// TIA Portal V17 export
// export: Created 2021-12-03T08:12:59.6189284Z, ExportSetting WithDefaults, DisplayName Totally Integrated Automation Portal, DisplayVersion V17, DisplayName TIA Portal Openness, DisplayVersion V17, DisplayName TIA Portal Version Control Interface, DisplayVersion V17, DisplayName STEP 7 Professional, DisplayVersion V17, DisplayName STEP 7 Safety, DisplayVersion V17, DisplayName WinCC Advanced, DisplayVersion V17
FUNCTION_BLOCK "FB_ScanSequence"   // FB70, GRAPH
VERSION : 0.1
// stored: AcknowledgeErrorsRequired true, AutoNumber false, CreateMinimizedDB false, IsIECCheckEnabled false, LanguageInNetworks LAD, LockOperatingMode false, PermanentILProcessingInMANMode false, SkipSteps false, UDAEnableTagReadback false, WithAlarmHandling true
   VAR_INPUT
      OFF_SQ { ExternalAccessible := 'False'; ExternalVisible := 'False'; ExternalWritable := 'False'} : Bool := false;   // Turn sequence off
      INIT_SQ { ExternalAccessible := 'False'; ExternalVisible := 'False'; ExternalWritable := 'False'} : Bool := false;   // Set sequence to initial state
      ACK_EF { ExternalAccessible := 'False'; ExternalVisible := 'False'; ExternalWritable := 'False'} : Bool := false;   // Acknowledge all errors and faults
      S_PREV { ExternalAccessible := 'False'; ExternalVisible := 'False'; ExternalWritable := 'False'} : Bool := false;   // Output previous step in parameter S_NO
      S_NEXT { ExternalAccessible := 'False'; ExternalVisible := 'False'; ExternalWritable := 'False'} : Bool := false;   // Indicate next step in parameter S_NO
      SW_AUTO { ExternalAccessible := 'False'; ExternalVisible := 'False'; ExternalWritable := 'False'} : Bool := false;   // Automatic mode
      SW_TAP { ExternalAccessible := 'False'; ExternalVisible := 'False'; ExternalWritable := 'False'} : Bool := false;   // Semiautomatic/switch with transition
      SW_TOP { ExternalAccessible := 'False'; ExternalVisible := 'False'; ExternalWritable := 'False'} : Bool := false;   // Semiautomatic/ignore transition
      SW_MAN { ExternalAccessible := 'False'; ExternalVisible := 'False'; ExternalWritable := 'False'} : Bool := false;   // Manual mode
      S_SEL { ExternalAccessible := 'False'; ExternalVisible := 'False'; ExternalWritable := 'False'} : Int := 0;   // Select step to be output to S_NO
      S_ON { ExternalAccessible := 'False'; ExternalVisible := 'False'; ExternalWritable := 'False'} : Bool := false;   // Activate step indicated in S_NO
      S_OFF { ExternalAccessible := 'False'; ExternalVisible := 'False'; ExternalWritable := 'False'} : Bool := false;   // Deactivate step indicated S_NO
      T_PUSH { ExternalAccessible := 'False'; ExternalVisible := 'False'; ExternalWritable := 'False'} : Bool := false;   // Enable transition to switch in semi automatic mode
   END_VAR
   VAR_OUTPUT
      S_NO { ExternalAccessible := 'False'; ExternalVisible := 'False'; ExternalWritable := 'False'} : Int := 0;   // Step number
      S_MORE { ExternalAccessible := 'False'; ExternalVisible := 'False'; ExternalWritable := 'False'} : Bool := false;   // More steps are available and can be shown in S_NO
      S_ACTIVE { ExternalAccessible := 'False'; ExternalVisible := 'False'; ExternalWritable := 'False'} : Bool := false;   // Step indicated in S_NO is active
      ERR_FLT { ExternalAccessible := 'False'; ExternalVisible := 'False'; ExternalWritable := 'False'} : Bool := false;   // Interlock or supervision group error
      AUTO_ON { ExternalAccessible := 'False'; ExternalVisible := 'False'; ExternalWritable := 'False'} : Bool := false;   // Automatic mode is active
      TAP_ON { ExternalAccessible := 'False'; ExternalVisible := 'False'; ExternalWritable := 'False'} : Bool := false;   // Semiautomatic mode/step with transition enabled
      TOP_ON { ExternalAccessible := 'False'; ExternalVisible := 'False'; ExternalWritable := 'False'} : Bool := false;   // Semiautomatic mode/ignore transition enabled
      MAN_ON { ExternalAccessible := 'False'; ExternalVisible := 'False'; ExternalWritable := 'False'} : Bool := false;   // Manual mode is active
   END_VAR
   VAR DB_SPECIFIC
      S_DISPLAY { ExternalAccessible := 'False'; ExternalVisible := 'False'; ExternalWritable := 'False'} : Int;   // Internal display of output parameter S_NO
      S_SEL_OLD { ExternalAccessible := 'False'; ExternalVisible := 'False'; ExternalWritable := 'False'} : Int;   // Previous value in S_SEL
      S_DISPIDX { ExternalAccessible := 'False'; ExternalVisible := 'False'; ExternalWritable := 'False'} : Byte;   // Index of the step in S_NO
      T_DISPIDX { ExternalAccessible := 'False'; ExternalVisible := 'False'; ExternalWritable := 'False'} : Byte;   // Index of the transition displayed in T_NO
      MOP { ExternalAccessible := 'False'; ExternalVisible := 'False'; ExternalWritable := 'False'} : Struct   // Mode
         AUTO { ExternalAccessible := 'False'; ExternalVisible := 'False'; ExternalWritable := 'False'} : Bool := true;   // Status: automatic mode
         MAN { ExternalAccessible := 'False'; ExternalVisible := 'False'; ExternalWritable := 'False'} : Bool := false;   // Status: manual mode
         TAP { ExternalAccessible := 'False'; ExternalVisible := 'False'; ExternalWritable := 'False'} : Bool := false;   // Status: semi automatic/switch with transition
         TOP { ExternalAccessible := 'False'; ExternalVisible := 'False'; ExternalWritable := 'False'} : Bool := false;   // Status: semi automatic/ignore transition
         ACK_S { ExternalAccessible := 'False'; ExternalVisible := 'False'; ExternalWritable := 'False'} : Bool := false;   // Request: acknowledge step at parameter S_NO
         REG_S { ExternalAccessible := 'False'; ExternalVisible := 'False'; ExternalWritable := 'False'} : Bool := false;   // Request: register step indicated in S_NO
         T_PREV { ExternalAccessible := 'False'; ExternalVisible := 'False'; ExternalWritable := 'False'} : Bool := false;   // Request: output previous valid transition in T_NO
         T_NEXT { ExternalAccessible := 'False'; ExternalVisible := 'False'; ExternalWritable := 'False'} : Bool := false;   // Request: output next valid transition in T_NO
         LOCK { ExternalAccessible := 'False'; ExternalVisible := 'False'; ExternalWritable := 'False'} : Bool := true;   // Status: interlocks activated
         SUP { ExternalAccessible := 'False'; ExternalVisible := 'False'; ExternalWritable := 'False'} : Bool := true;   // Status: supervisions activated
         ACKREQ { ExternalAccessible := 'False'; ExternalVisible := 'False'; ExternalWritable := 'False'} : Bool := true;   // Status: acknowledgment required
         SSKIP { ExternalAccessible := 'False'; ExternalVisible := 'False'; ExternalWritable := 'False'} : Bool := false;   // Status: "Skip steps" enabled
         OFF { ExternalAccessible := 'False'; ExternalVisible := 'False'; ExternalWritable := 'False'} : Bool := false;   // Request: deactivate all steps
         INIT { ExternalAccessible := 'False'; ExternalVisible := 'False'; ExternalWritable := 'False'} : Bool := true;   // Request: set sequence to initial state
         HALT { ExternalAccessible := 'False'; ExternalVisible := 'False'; ExternalWritable := 'False'} : Bool := false;   // Status: sequence halted
         TMS_HALT { ExternalAccessible := 'False'; ExternalVisible := 'False'; ExternalWritable := 'False'} : Bool := false;   // Status: all internal timers held
         OPS_ZERO { ExternalAccessible := 'False'; ExternalVisible := 'False'; ExternalWritable := 'False'} : Bool := false;   // Status: set all operands processed with N, L, D instructions to 0
         SACT_DISP { ExternalAccessible := 'False'; ExternalVisible := 'False'; ExternalWritable := 'False'} : Bool := true;   // Status: display active steps only
         SEF_DISP { ExternalAccessible := 'False'; ExternalVisible := 'False'; ExternalWritable := 'False'} : Bool := false;   // Status: display only steps with errors and disrupted steps
         SALL_DISP { ExternalAccessible := 'False'; ExternalVisible := 'False'; ExternalWritable := 'False'} : Bool := false;   // Status: display all steps
         S_PREV { ExternalAccessible := 'False'; ExternalVisible := 'False'; ExternalWritable := 'False'} : Bool := false;   // Request: output previous step to S_NO
         S_NEXT { ExternalAccessible := 'False'; ExternalVisible := 'False'; ExternalWritable := 'False'} : Bool := false;   // Request: Output next step at S_NO parameter
         S_SELOK { ExternalAccessible := 'False'; ExternalVisible := 'False'; ExternalWritable := 'False'} : Bool := false;   // Request: output step number from S_SEL to S_NO
         S_ON { ExternalAccessible := 'False'; ExternalVisible := 'False'; ExternalWritable := 'False'} : Bool := false;   // Request: activate step indicated in S_NO
         S_OFF { ExternalAccessible := 'False'; ExternalVisible := 'False'; ExternalWritable := 'False'} : Bool := false;   // Request: deactivate step at parameter S_NO
         T_PUSH { ExternalAccessible := 'False'; ExternalVisible := 'False'; ExternalWritable := 'False'} : Bool := false;   // Request: transition switching enabled
         REG { ExternalAccessible := 'False'; ExternalVisible := 'False'; ExternalWritable := 'False'} : Bool := false;   // Request: register all interlock and supervision errors
         ACK { ExternalAccessible := 'False'; ExternalVisible := 'False'; ExternalWritable := 'False'} : Bool := false;   // Request: acknowledge all interlock and supervision errors
         IL_PERM { ExternalAccessible := 'False'; ExternalVisible := 'False'; ExternalWritable := 'False'} : Bool := false;   // Status: permanent processing of all interlocks
         T_PERM { ExternalAccessible := 'False'; ExternalVisible := 'False'; ExternalWritable := 'False'} : Bool := false;   // Status: permanent processing of all transitions
         ILP_MAN { ExternalAccessible := 'False'; ExternalVisible := 'False'; ExternalWritable := 'False'} : Bool := false;   // Status: permanent processing of all interlocks in manual mode
      END_STRUCT;
      TICKS { ExternalAccessible := 'False'; ExternalVisible := 'False'; ExternalWritable := 'False'} : Struct   // Clock speeds
         DELTA { ExternalAccessible := 'False'; ExternalVisible := 'False'; ExternalWritable := 'False'} : Time := T#0ms;   // Time difference between cycles
         OLD { ExternalAccessible := 'False'; ExternalVisible := 'False'; ExternalWritable := 'False'} : Time := T#0ms;   // 10 ms clock counter value in last cycle
         NEW { ExternalAccessible := 'False'; ExternalVisible := 'False'; ExternalWritable := 'False'} : Time := T#0ms;   // 10 ms clock counter value in this cycle
      END_STRUCT;
      SQ_FLAGS { ExternalAccessible := 'False'; ExternalVisible := 'False'; ExternalWritable := 'False'} : Struct   // Sequence bit memory
         ERR_FLT { ExternalAccessible := 'False'; ExternalVisible := 'False'; ExternalWritable := 'False'} : Bool := false;   // Interlock and supervision group error
         ERROR { ExternalAccessible := 'False'; ExternalVisible := 'False'; ExternalWritable := 'False'} : Bool := false;   // Interlock group error
         FAULT { ExternalAccessible := 'False'; ExternalVisible := 'False'; ExternalWritable := 'False'} : Bool := false;   // Supervision group error
         RT_FAIL { ExternalAccessible := 'False'; ExternalVisible := 'False'; ExternalWritable := 'False'} : Bool := false;   // Runtime error
         NO_SNO { ExternalAccessible := 'False'; ExternalVisible := 'False'; ExternalWritable := 'False'} : Bool := false;   // Requested step number not found
         NF_OFL { ExternalAccessible := 'False'; ExternalVisible := 'False'; ExternalWritable := 'False'} : Bool := false;   // Overflow: too many ON or OFF requests
         SA_OFL { ExternalAccessible := 'False'; ExternalVisible := 'False'; ExternalWritable := 'False'} : Bool := false;   // Overflow: too many steps active
         TV_OFL { ExternalAccessible := 'False'; ExternalVisible := 'False'; ExternalWritable := 'False'} : Bool := false;   // Overflow: too many valid transitions
         MSG_OFL { ExternalAccessible := 'False'; ExternalVisible := 'False'; ExternalWritable := 'False'} : Bool := false;   // Overflow: not enough system resources for ALARM_S
         NO_SWI { ExternalAccessible := 'False'; ExternalVisible := 'False'; ExternalWritable := 'False'} : Bool := false;   // Do not switch in this cycle
         CYC_OP { ExternalAccessible := 'False'; ExternalVisible := 'False'; ExternalWritable := 'False'} : Bool := false;   // Cyclic execution of the sequence after initialization
         AS_MSG { ExternalAccessible := 'False'; ExternalVisible := 'False'; ExternalWritable := 'False'} : Bool := true;   // Alarms during runtime enabled or disabled by instruction
         AS_SEND { ExternalAccessible := 'False'; ExternalVisible := 'False'; ExternalWritable := 'False'} : Bool := false;   // Send alarms from WR_USMSG or only enter in diagnostics buffer
         SQ_BUSY { ExternalAccessible := 'False'; ExternalVisible := 'False'; ExternalWritable := 'False'} : Bool := false;   // Internal edge memory bit for sequence processing
         SA_BUSY { ExternalAccessible := 'False'; ExternalVisible := 'False'; ExternalWritable := 'False'} : Bool := false;   // Internal edge memory bit for sequence processing
         AS_SIG { ExternalAccessible := 'False'; ExternalVisible := 'False'; ExternalWritable := 'False'} : Bool := false;   // Edge memory bit for alarms from Alarm_S and Alarm_SQ
      END_STRUCT;
   END_VAR
BEGIN
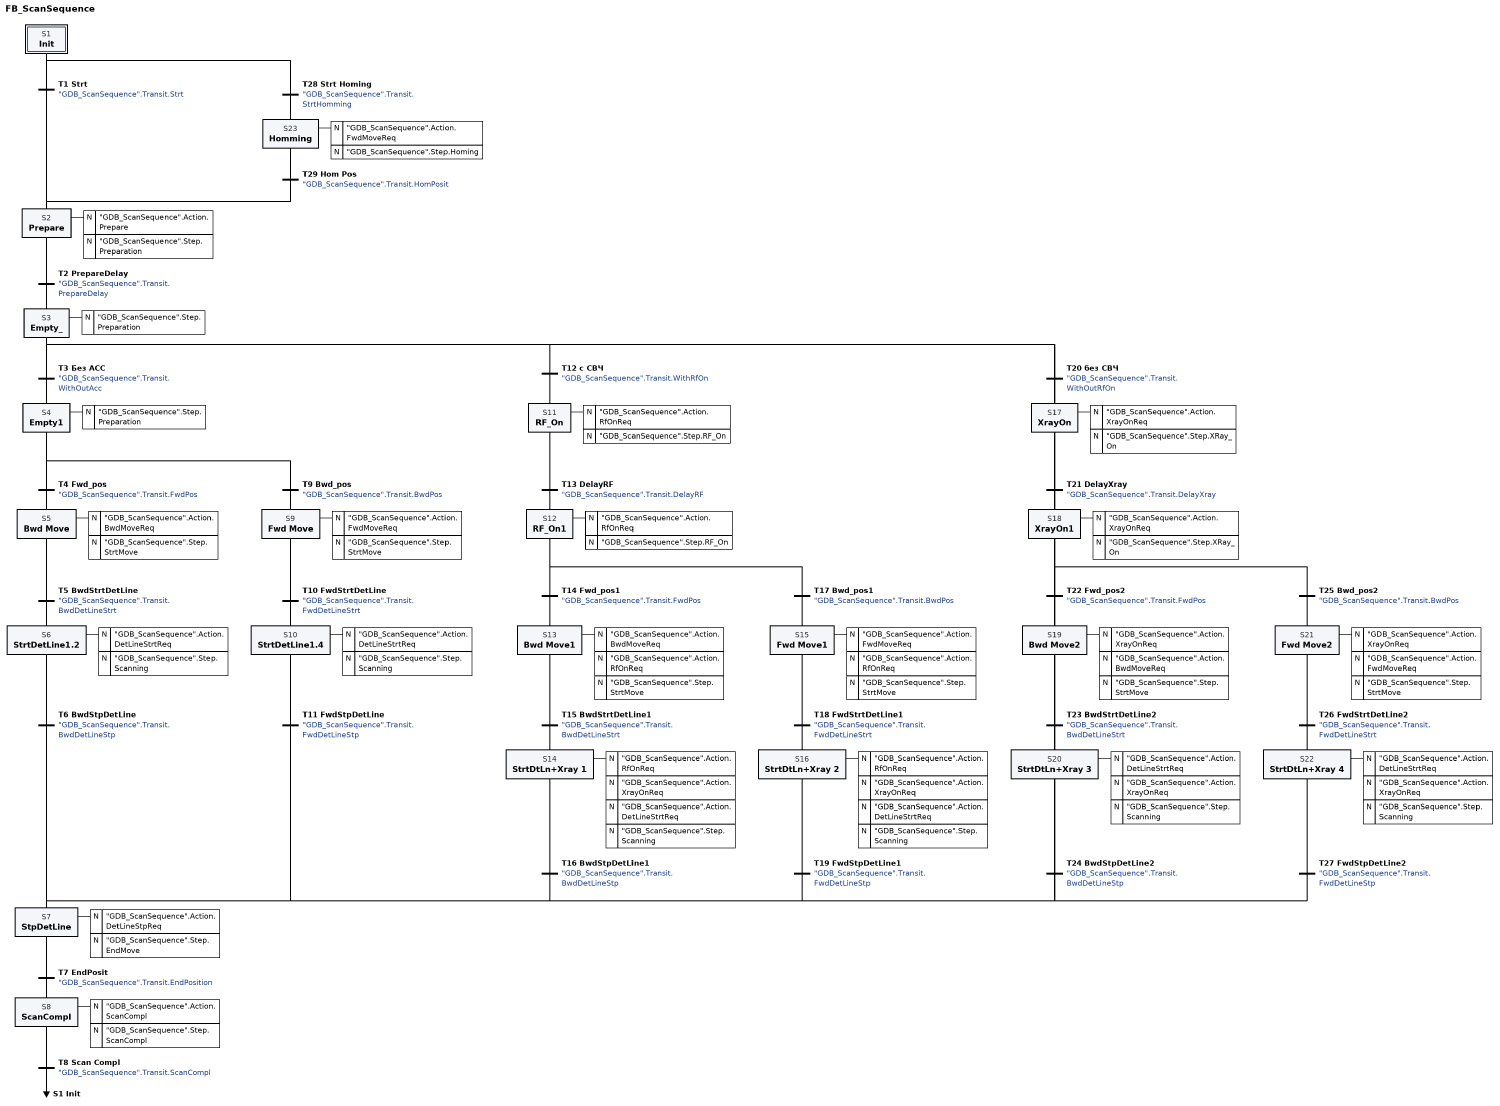
   // sequencer 1
   INITIAL_STEP Init:   // S1
   END_STEP
   TRANSITION Strt FROM Init TO Prepare   // T1
      := "GDB_ScanSequence".Transit.Strt;
   END_TRANSITION
   TRANSITION "Strt Homing" FROM Init TO Homming   // T28
      := "GDB_ScanSequence".Transit.StrtHomming;
   END_TRANSITION
   STEP Prepare:   // S2
              N    "GDB_ScanSequence".Action.Prepare
              N    "GDB_ScanSequence".Step.Preparation
   END_STEP
   TRANSITION PrepareDelay FROM Prepare TO Empty_   // T2
      := "GDB_ScanSequence".Transit.PrepareDelay;
   END_TRANSITION
   STEP Empty1:   // S4
              N    "GDB_ScanSequence".Step.Preparation
   END_STEP
   TRANSITION Fwd_pos FROM Empty1 TO "Bwd Move"   // T4
      := "GDB_ScanSequence".Transit.FwdPos;
   END_TRANSITION
   TRANSITION Bwd_pos FROM Empty1 TO "Fwd Move"   // T9
      := "GDB_ScanSequence".Transit.BwdPos;
   END_TRANSITION
   STEP "Bwd Move1":   // S13
              N    "GDB_ScanSequence".Action.BwdMoveReq
              N    "GDB_ScanSequence".Action.RfOnReq
              N    "GDB_ScanSequence".Step.StrtMove
   END_STEP
   TRANSITION BwdStrtDetLine1 FROM "Bwd Move1" TO "StrtDtLn+Xray 1"   // T15
      := "GDB_ScanSequence".Transit.BwdDetLineStrt;
   END_TRANSITION
   STEP "Bwd Move":   // S5
              N    "GDB_ScanSequence".Action.BwdMoveReq
              N    "GDB_ScanSequence".Step.StrtMove
   END_STEP
   TRANSITION BwdStrtDetLine FROM "Bwd Move" TO "StrtDetLine1.2"   // T5
      := "GDB_ScanSequence".Transit.BwdDetLineStrt;
   END_TRANSITION
   STEP "Fwd Move":   // S9
              N    "GDB_ScanSequence".Action.FwdMoveReq
              N    "GDB_ScanSequence".Step.StrtMove
   END_STEP
   TRANSITION FwdStrtDetLine FROM "Fwd Move" TO "StrtDetLine1.4"   // T10
      := "GDB_ScanSequence".Transit.FwdDetLineStrt;
   END_TRANSITION
   STEP "StrtDetLine1.2":   // S6
              N    "GDB_ScanSequence".Action.DetLineStrtReq
              N    "GDB_ScanSequence".Step.Scanning
   END_STEP
   TRANSITION BwdStpDetLine FROM "StrtDetLine1.2" TO StpDetLine   // T6
      := "GDB_ScanSequence".Transit.BwdDetLineStp;
   END_TRANSITION
   STEP "StrtDetLine1.4":   // S10
              N    "GDB_ScanSequence".Action.DetLineStrtReq
              N    "GDB_ScanSequence".Step.Scanning
   END_STEP
   TRANSITION FwdStpDetLine FROM "StrtDetLine1.4" TO StpDetLine   // T11
      := "GDB_ScanSequence".Transit.FwdDetLineStp;
   END_TRANSITION
   STEP StpDetLine:   // S7
              N    "GDB_ScanSequence".Action.DetLineStpReq
              N    "GDB_ScanSequence".Step.EndMove
   END_STEP
   TRANSITION EndPosit FROM StpDetLine TO ScanCompl   // T7
      := "GDB_ScanSequence".Transit.EndPosition;
   END_TRANSITION
   STEP ScanCompl:   // S8
              N    "GDB_ScanSequence".Action.ScanCompl
              N    "GDB_ScanSequence".Step.ScanCompl
   END_STEP
   TRANSITION "Scan Compl" FROM ScanCompl TO Init   // T8, jump
      := "GDB_ScanSequence".Transit.ScanCompl;
   END_TRANSITION
   STEP "Fwd Move1":   // S15
              N    "GDB_ScanSequence".Action.FwdMoveReq
              N    "GDB_ScanSequence".Action.RfOnReq
              N    "GDB_ScanSequence".Step.StrtMove
   END_STEP
   TRANSITION FwdStrtDetLine1 FROM "Fwd Move1" TO "StrtDtLn+Xray 2"   // T18
      := "GDB_ScanSequence".Transit.FwdDetLineStrt;
   END_TRANSITION
   STEP RF_On:   // S11
              N    "GDB_ScanSequence".Action.RfOnReq
              N    "GDB_ScanSequence".Step.RF_On
   END_STEP
   TRANSITION DelayRF FROM RF_On TO RF_On1   // T13
      := "GDB_ScanSequence".Transit.DelayRF;
   END_TRANSITION
   STEP "StrtDtLn+Xray 1":   // S14
              N    "GDB_ScanSequence".Action.RfOnReq
              N    "GDB_ScanSequence".Action.XrayOnReq
              N    "GDB_ScanSequence".Action.DetLineStrtReq
              N    "GDB_ScanSequence".Step.Scanning
   END_STEP
   TRANSITION BwdStpDetLine1 FROM "StrtDtLn+Xray 1" TO StpDetLine   // T16
      := "GDB_ScanSequence".Transit.BwdDetLineStp;
   END_TRANSITION
   STEP "StrtDtLn+Xray 2":   // S16
              N    "GDB_ScanSequence".Action.RfOnReq
              N    "GDB_ScanSequence".Action.XrayOnReq
              N    "GDB_ScanSequence".Action.DetLineStrtReq
              N    "GDB_ScanSequence".Step.Scanning
   END_STEP
   TRANSITION FwdStpDetLine1 FROM "StrtDtLn+Xray 2" TO StpDetLine   // T19
      := "GDB_ScanSequence".Transit.FwdDetLineStp;
   END_TRANSITION
   STEP RF_On1:   // S12
              N    "GDB_ScanSequence".Action.RfOnReq
              N    "GDB_ScanSequence".Step.RF_On
   END_STEP
   TRANSITION Fwd_pos1 FROM RF_On1 TO "Bwd Move1"   // T14
      := "GDB_ScanSequence".Transit.FwdPos;
   END_TRANSITION
   TRANSITION Bwd_pos1 FROM RF_On1 TO "Fwd Move1"   // T17
      := "GDB_ScanSequence".Transit.BwdPos;
   END_TRANSITION
   STEP "Bwd Move2":   // S19
              N    "GDB_ScanSequence".Action.XrayOnReq
              N    "GDB_ScanSequence".Action.BwdMoveReq
              N    "GDB_ScanSequence".Step.StrtMove
   END_STEP
   TRANSITION BwdStrtDetLine2 FROM "Bwd Move2" TO "StrtDtLn+Xray 3"   // T23
      := "GDB_ScanSequence".Transit.BwdDetLineStrt;
   END_TRANSITION
   STEP "Fwd Move2":   // S21
              N    "GDB_ScanSequence".Action.XrayOnReq
              N    "GDB_ScanSequence".Action.FwdMoveReq
              N    "GDB_ScanSequence".Step.StrtMove
   END_STEP
   TRANSITION FwdStrtDetLine2 FROM "Fwd Move2" TO "StrtDtLn+Xray 4"   // T26
      := "GDB_ScanSequence".Transit.FwdDetLineStrt;
   END_TRANSITION
   STEP XrayOn:   // S17
              N    "GDB_ScanSequence".Action.XrayOnReq
              N    "GDB_ScanSequence".Step.XRay_On
   END_STEP
   TRANSITION DelayXray FROM XrayOn TO XrayOn1   // T21
      := "GDB_ScanSequence".Transit.DelayXray;
   END_TRANSITION
   STEP "StrtDtLn+Xray 3":   // S20
              N    "GDB_ScanSequence".Action.DetLineStrtReq
              N    "GDB_ScanSequence".Action.XrayOnReq
              N    "GDB_ScanSequence".Step.Scanning
   END_STEP
   TRANSITION BwdStpDetLine2 FROM "StrtDtLn+Xray 3" TO StpDetLine   // T24
      := "GDB_ScanSequence".Transit.BwdDetLineStp;
   END_TRANSITION
   STEP "StrtDtLn+Xray 4":   // S22
              N    "GDB_ScanSequence".Action.DetLineStrtReq
              N    "GDB_ScanSequence".Action.XrayOnReq
              N    "GDB_ScanSequence".Step.Scanning
   END_STEP
   TRANSITION FwdStpDetLine2 FROM "StrtDtLn+Xray 4" TO StpDetLine   // T27
      := "GDB_ScanSequence".Transit.FwdDetLineStp;
   END_TRANSITION
   STEP XrayOn1:   // S18
              N    "GDB_ScanSequence".Action.XrayOnReq
              N    "GDB_ScanSequence".Step.XRay_On
   END_STEP
   TRANSITION Fwd_pos2 FROM XrayOn1 TO "Bwd Move2"   // T22
      := "GDB_ScanSequence".Transit.FwdPos;
   END_TRANSITION
   TRANSITION Bwd_pos2 FROM XrayOn1 TO "Fwd Move2"   // T25
      := "GDB_ScanSequence".Transit.BwdPos;
   END_TRANSITION
   STEP Homming:   // S23
              N    "GDB_ScanSequence".Action.FwdMoveReq
              N    "GDB_ScanSequence".Step.Homing
   END_STEP
   TRANSITION "Hom Pos" FROM Homming TO Prepare   // T29
      := "GDB_ScanSequence".Transit.HomPosit;
   END_TRANSITION
   STEP Empty_:   // S3
              N    "GDB_ScanSequence".Step.Preparation
   END_STEP
   TRANSITION "Без ACC" FROM Empty_ TO Empty1   // T3
      := "GDB_ScanSequence".Transit.WithOutAcc;
   END_TRANSITION
   TRANSITION "с СВЧ" FROM Empty_ TO RF_On   // T12
      := "GDB_ScanSequence".Transit.WithRfOn;
   END_TRANSITION
   TRANSITION "без СВЧ" FROM Empty_ TO XrayOn   // T20
      := "GDB_ScanSequence".Transit.WithOutRfOn;
   END_TRANSITION
END_FUNCTION_BLOCK
